PROGRAM Taks_2
VAR
	need: INT;
	timer: TON;	
	Wait5s: Wait;
END_VAR

//GVL.need_1 := 0;
IF GVL.need_1 < 100 THEN
	timer(IN := TRUE, PT := T#1S);
	IF timer.Q = TRUE THEN
		gvl.need_1 := gvl.need_1+1;	
		timer(IN := FALSE);
	END_IF
END_IF

END_PROGRAM

(* stored: Version 1.1.0.1, ProductVersion 3.1.4024.15
   POU Taks_2: Id {3f954ceb-7654-4c46-82ae-7c4cd977fac6}, SpecialFunc None *)
